INTERFACE I_EnumeratorConnectionUpdater

METHOD PUBLIC AddConnection
VAR_INPUT
	EnumeratorConnection : I_EnumeratorConnection;
END_VAR
END_METHOD

METHOD PUBLIC RemoveConnection
VAR_INPUT
	EnumeratorConnection : I_EnumeratorConnection;
END_VAR
END_METHOD

END_INTERFACE

(* stored: Version 1.1.0.1, ProductVersion 3.1.4024.12
   Itf I_EnumeratorConnectionUpdater: Id {0c564cf9-4b79-46e7-91a3-6e2917816de8}
   Method AddConnection: Id {32da9560-45b6-4d5c-8d96-c30aa3ec4a5e}
   Method RemoveConnection: Id {35c9f0b7-ebac-4c58-96ff-ecff54fc3657} *)
